# EPICS substitutions: evrSupport/Db/ioc/IOC-IN20-RF01bsa.substitutions
# BSA records
#
# One per device:
# Please check the HOPR,LOPR,PREC,ADEL,MDEL values provided in bsaPHASEdef.db!
file bsaPHASEdef.db {
#      Device               ,loc'n , IOC  , system, Attribute
  pattern {DEVICE           , LOC  ,  UN  , SYS   , ATRB  }
	  { LLRF:IN20:1         , IN20 , RF01 , SYS0  , REF_P }
	  { LASR:IN20:1         , IN20 , RF01 , SYS0  , P     }
	  { GUN:IN20:1          , IN20 , RF01 , SYS0  , RF_P  }
	  { GUN:IN20:2          , IN20 , RF01 , SYS0  , RF_P  }
	  { ACCL:IN20:300       , IN20 , RF01 , SYS0  , L0A_P }
	  { ACCL:IN20:400       , IN20 , RF01 , SYS0  , LOB_P }
	  { TCAV:IN20:490       , IN20 , RF01 , SYS0  , P     }
	  { PCAV:IN20:365       , IN20 , RF01 , SYS0  , P     }
}
# One per device:
# Please check the HOPR,LOPR,PREC,ADEL,MDEL values provided in bsaAMPLEdef.db!
file bsaAMPLEdef.db {
#      Device               ,loc'n , IOC  ,system , Attribute
  pattern {DEVICE           , LOC  ,  UN  , SYS   , ATRB  }
	  { LLRF:IN20:1         , IN20 , RF01 , SYS0  , REF_A }
	  { LASR:IN20:1         , IN20 , RF01 , SYS0  , A     }
	  { GUN:IN20:1          , IN20 , RF01 , SYS0  , RF_A  }
	  { GUN:IN20:2          , IN20 , RF01 , SYS0  , RF_A  }
	  { ACCL:IN20:300       , IN20 , RF01 , SYS0  , L0A_A }
	  { ACCL:IN20:400       , IN20 , RF01 , SYS0  , LOB_A }
	  { TCAV:IN20:490       , IN20 , RF01 , SYS0  , A     }
	  { PCAV:IN20:365       , IN20 , RF01 , SYS0  , A     }
